Fanuc KAREL source: kb00101.KL

-- PROVISIONAL review KL for V1013-1; original PC SHA256 d0026231e901a493f0f4456b1ac0d72ae2b8e979c12a6c2d8fab612eba905386
-- Incomplete behavior may be omitted. Consult companion uncertainty JSON. Do not deploy.
PROGRAM KB00101
%NOLOCKGROUP
BEGIN
  -- UNRESOLVED_PC offsets 5-12; opcodes 9D,23
  -- UNRESOLVED_PC offsets 17-26; opcodes 3F,75
  -- UNRESOLVED_PC offsets 31-38; opcodes 9D,23
  -- UNRESOLVED_PC offsets 43-50; opcodes 9D,23
  -- UNRESOLVED_PC offsets 55-62; opcodes 9D,23
  -- UNRESOLVED_PC offsets 67-74; opcodes 9D,23
  -- UNRESOLVED_PC offsets 79-86; opcodes 9D,23
  -- UNRESOLVED_PC offsets 91-98; opcodes 9D,23
  -- UNRESOLVED_PC offsets 103-110; opcodes 9D,23
  -- UNRESOLVED_PC offsets 115-181; opcodes 27,22,22,2A,22,22,22,22,22,22,22,22,31
  -- UNRESOLVED_PC offsets 186-190; opcodes 7F
END KB00101
